FUNCTION_BLOCK ReadyUnifiedProgramState EXTENDS ReadyProgramState
VAR
	{attribute 'OPC.UA.DA' := '0'}
	_ClassName : STRING := __POUNAME();
END_VAR

{attribute 'monitoring' := 'call'}
PROPERTY ClassName : STRING
GET
ClassName := _ClassName;
END_GET
END_PROPERTY

END_FUNCTION_BLOCK

(* stored: Version 1.1.0.1
   POU ReadyUnifiedProgramState: Id {ab67e381-18c6-411a-906f-10d5360c3e19}, SpecialFunc None
   Property ClassName: Id {2c057c0a-2343-42b1-8e66-8a3c0760d7e1}
   Get Get: Id {e0dd91e4-8a2a-47cc-b237-2ff470d4277d} *)
